TYPE ST_CylinderX_Config :
    STRUCT
        ExtendTime  : LREAL;
        RetractTime : LREAL;
    END_STRUCT
END_TYPE

(* stored: Version 1.1.0.1, ProductVersion 3.1.4024.15
   DUT ST_CylinderX_Config: Id {982f8ba7-035b-0308-0ff1-2ac43301b0e7} *)
